ABB RobotStudio station: 20msyo2026.rsstnx

Station 20msyo2026 (saved by RobotStudio 25.5.11605.0)
Controller IRB140_6_81
  mechanical unit ROB_1: IRB140_6_81_C_03, 6 joints, base frame (0, 0, 0) mm
Layout (positions relative to the parent item):
  - IRB140_6_81_C_03 [mechanism, from %ABB.RobotStudio.Models.IRB140%\IRB140_6_81_C_G_03.rslib] at (0, 0, 0) mm; joint values [-0.0997, 0.456, -0.2852, 0, 1.4001, -2.8486] (rad or m)
  - Part_3 [part], size 10 x 10 x 10 mm
  - Part_7 [part], size 7 x 7 x 100 mm
  - Mesa [part], size 365 x 405 x 340 mm
  - perno [part] at (1000, -190, 228.67) mm, rotated rx 90 ry 0 rz 180 deg, size 20 x 100 x 20 mm
  - Pinza [mechanism] at (600, -60, 545.67) mm, rotated rx -180 ry 0 rz -22.5 deg
      TCP Pinza at (0, 0, 137) mm, rotated rx 0 ry 0 rz -22.5 deg
      links: Dummy
Attachment: Pinza is attached to IRB140_6_81_C_03 / Link6
Attachment: mesa is attached to Mesa
Attachment: perno is attached to Pinza / Dummy
EventTableEntry 2368: ActivationMode=2, Cyclic=false, Group=, Trigger=DO_Pinza 2369, Actions=[EventTableActionAttach 2370], Comment=
EventTableTriggerIO 2369: Operator=0, IOValue=[1], IRC5Controller=? -1, SignalSource=IRB140_6_81 1261
EventTableActionAttach 2370: MountObject=false, FlangeIndext=0, FindNearest=false, AttachmentParent=Pinza 2362, AttachmentChild=perno 2358, Offset=[X=1, Y=0, Z=0, W=0, X=0, Y=1, Z=0, W=0, X=0, Y=0, Z=1, W=0, X=0, Y=0, Z=0, W=1]
EventTableEntry 2371: ActivationMode=2, Cyclic=false, Group=, Trigger=DO_Pinza 2372, Actions=[EventTableActionDetach 2373], Comment=
EventTableTriggerIO 2372: Operator=0, IOValue=[0], IRC5Controller=? -1, SignalSource=IRB140_6_81 1261
EventTableActionDetach 2373: AttachmentParent=Pinza 2362, AttachmentChild=perno 2358
Collision set CollisionSet_2: perno against Mesa, near miss 0.005 m
EventTableTriggerIO 2424: Operator=0, IOValue=[1], IRC5Controller=? -1, SignalSource=IRB140_6_81 1261
EventTableTriggerIO 2425: Operator=0, IOValue=[1], IRC5Controller=? -1, SignalSource=IRB140_6_81 1261
EventTableTriggerIO 2426: Operator=0, IOValue=[0], IRC5Controller=? -1, SignalSource=IRB140_6_81 1261
EventTableTriggerIO 2427: Operator=0, IOValue=[0], IRC5Controller=? -1, SignalSource=IRB140_6_81 1261
EventTableTriggerIO 2428: Operator=0, IOValue=[1], IRC5Controller=? -1, SignalSource=IRB140_6_81 1261
EventTableTriggerIO 2429: Operator=0, IOValue=[1], IRC5Controller=? -1, SignalSource=IRB140_6_81 1261
EventTableTriggerIO 2430: Operator=0, IOValue=[1], IRC5Controller=? -1, SignalSource=IRB140_6_81 1261
EventTableTriggerIO 2431: Operator=0, IOValue=[0], IRC5Controller=? -1, SignalSource=IRB140_6_81 1261
EventTableTriggerIO 2432: Operator=0, IOValue=[0], IRC5Controller=? -1, SignalSource=IRB140_6_81 1261
EventTableTriggerIO 2433: Operator=0, IOValue=[0], IRC5Controller=? -1, SignalSource=IRB140_6_81 1261
EventTableTriggerIO 2518: Operator=0, IOValue=[1], IRC5Controller=? -1, SignalSource=IRB140_6_81 1261
EventTableTriggerIO 2519: Operator=0, IOValue=[1], IRC5Controller=? -1, SignalSource=IRB140_6_81 1261
EventTableTriggerIO 2520: Operator=0, IOValue=[1], IRC5Controller=? -1, SignalSource=IRB140_6_81 1261
EventTableTriggerIO 2521: Operator=0, IOValue=[0], IRC5Controller=? -1, SignalSource=IRB140_6_81 1261
EventTableTriggerIO 2522: Operator=0, IOValue=[0], IRC5Controller=? -1, SignalSource=IRB140_6_81 1261
EventTableTriggerIO 2523: Operator=0, IOValue=[0], IRC5Controller=? -1, SignalSource=IRB140_6_81 1261
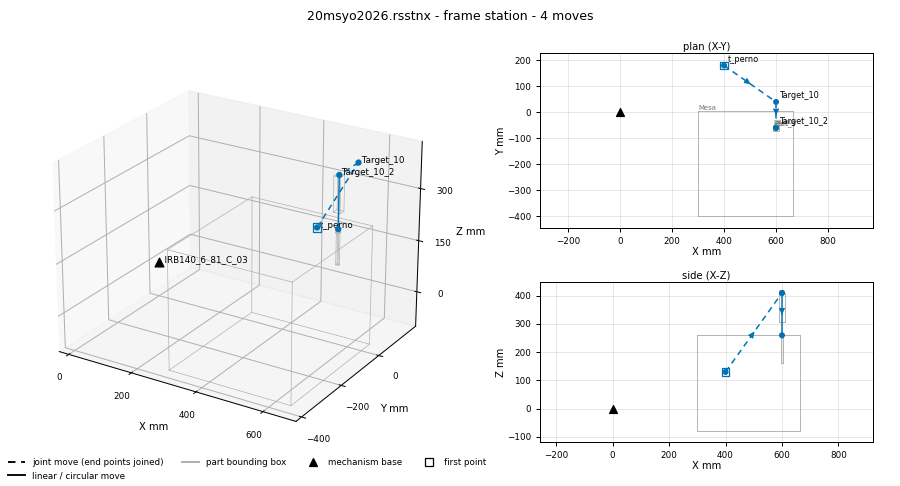
[picture p0: tool path of 20msyo2026.rsstnx in frame station, 4 of 4 moves have a stored position in this frame; points joined in program order, loops and branches not executed]
Targets, tools, work objects and paths stored in the station, written as RAPID:
! task T_ROB1
MODULE CalibData
  PERS tooldata Pinza:=[TRUE,[[0,0,137],[0.98078528,0,0,-0.195090322]],[0.5,[0,0,100],[1,0,0,0],0,0,0]];
  TASK PERS wobjdata mesa:=[FALSE,TRUE,"",[[665,5,260],[0,0,0,1]],[[0,0,0],[1,0,0,0]]];
  PERS wobjdata perno:=[FALSE,TRUE,"",[[400,180,130],[0.707106781,-0.707106781,0,0]],[[0,0,0],[1,0,0,0]]];
ENDMODULE

! task T_ROB1
MODULE Module1
  CONST robtarget t_agujero:=[[65,65,0],[0,0,1,0],[0,0,0,0],[9E+09,9E+09,9E+09,9E+09,9E+09,9E+09]];
  CONST robtarget t_perno:=[[0,0,0],[0,0,1,0],[0,0,0,0],[9E+09,9E+09,9E+09,9E+09,9E+09,9E+09]];
  CONST robtarget Target_10:=[[65,-35,150],[0,0,1,0],[-1,0,-2,0],[9E+09,9E+09,9E+09,9E+09,9E+09,9E+09]];
  CONST robtarget Target_10_2:=[[65,65,150],[0,0,1,0],[-1,0,-2,0],[9E+09,9E+09,9E+09,9E+09,9E+09,9E+09]];
  PROC Path_10()
    MoveL t_perno,v100,fine,Pinza\WObj:=perno;
    WaitTime \InPos,1;
    SetDO DO_Pinza,1;
    MoveJ Target_10,v100,z10,Pinza\WObj:=mesa;
    MoveJ Target_10_2,v100,z10,Pinza\WObj:=mesa;
    MoveL t_agujero,v30,fine,Pinza\WObj:=mesa;
    SetDO DO_Pinza,0;
  ENDPROC
ENDMODULE

